TYPE (* IEC61131-3, Table 14#5 *)
  (* Standard: 1131-3 *)
  (* Version 0.0, 1/8/2024, Cheyan, Schneider Electric, Template *)
  PACKAGE Main;
  {SET_ATTRIBUTE(nxtDataType, Lp5NebPSNARI2wwB7co/OJ7bm7Z6XnroHaJ9upnY2JiKs/1FJEdQUGp8i6Yee8lC5/PwtQPe9I9G+N2G/wSstA==)}
  validity : (
    good,
    invalid,
    reserved,
    questionable
  );
END_TYPE
